// SIMATIC STEP 7 (V5.x) project S_desbobinado
// CPU: CPU312(1)
// station: P_ADR_BUS
// station: Hardware
// station: Equipo SIMATIC 300
// program: Programa S7(1)

SYMBOL_TABLE
"CONTADOR"	C 1	COUNTER
"DESBOBINADO"	FB 1	FB 1	// Función que se encarga del desbobinado
"SENSOR"	I 124.0	BOOL
"PRESENCIA"	I 124.1	BOOL
"BIT_DE_TRABAJO"	I 124.2	BOOL
"START"	I 124.3	BOOL
"STOP"	I 124.4	BOOL
"BAJAR_CONT"	I 124.5	BOOL
"LOAD_CONT"	I 124.6	BOOL
"Cycle Execution"	OB 1	OB 1
"PLANCHAS"	PIW 651	WORD
"CENTRO"	PIW 751	INT
"MCENTRO"	PIW 800	INT
"ABRIRMCENTRO"	Q 100.1	BOOL
"DESBOBINAR"	Q 100.2	BOOL
"BIT_OK"	Q 100.3	BOOL
"BIT_ERROR"	Q 100.4	BOOL
"STBY"	Q 100.5	BOOL
END_SYMBOL_TABLE

FUNCTION_BLOCK "DESBOBINADO"	// FB 1
TITLE = DESBOBINADO
VERSION : 0.1
VAR_INPUT
  SENSOR : BOOL ;
  PRESENCIA : BOOL ;
  CENTRO : INT ;
  bit_de_trabajo : BOOL ;
  MCENTRO : INT ;
  Contador : COUNTER ;
  START : BOOL ;
  PLANCHAS : WORD  := W#16#100;
END_VAR
VAR_OUTPUT
  ABRIRMCENTRO : BOOL ;
  DESBOBINAR : BOOL ;
  STBY : BOOL ;
END_VAR
VAR
  x31 : BOOL ;
  x32 : BOOL ;
  x33 : BOOL ;
  x34 : BOOL ;
  s1 : BOOL ;
  FP_Bit_Tr : BOOL ;
  x30 : BOOL ;
  FP_PRESENCIA : BOOL ;
  FP_BDT : BOOL ;
  FP_START : BOOL ;
END_VAR
VAR_TEMP
  watchdog_master : BOOL ;
END_VAR
BEGIN
NETWORK
TITLE = Arranque
      SET;
      A     #bit_de_trabajo;
      FP    #FP_BDT;
      S     #x30;
      R     #x31;
      R     #x32;
      R     #x33;
      R     #x34;
      R     #s1;
NETWORK
TITLE = x31 a x32
//Comparacion medida centro con medida nominal del centro para pasar de x31 a x32
      A     #x31;
      A(;
      L     #CENTRO;
      L     #MCENTRO;
      ==R;
      );
      R     #x31;
      S     #x32;
NETWORK
TITLE = x32 a x33
//Presencia detecta que la plancha esta en posicion para empezar el proceso de 
//desbobinado-cizallado
      A     #x32;
      A     #PRESENCIA;
      FP    #FP_PRESENCIA;
      R     #x32;
      S     #x33;
NETWORK
TITLE = x33 a x34
//Detecta que la plancha esta lista para ser cizallada
      A     #x33;
      A     #SENSOR;
      R     #x33;
      S     #x34;
NETWORK
TITLE = x34 a x33
//si el contador no ha acabado
      A     #x34;
      T     LD 1;
      TAK;
      T     LD 5;
      L     #Contador;
      T     LW 9;
      L     LD 5;
      L     LD 1;
      A     C [LW 9];
      AN    #SENSOR;
      R     #x34;
      S     #x33;
NETWORK
TITLE = x34 a s1
//si el contador ha cabado
      A     #x34;
      T     LD 1;
      TAK;
      T     LD 5;
      L     #Contador;
      T     LW 9;
      L     LD 5;
      L     LD 1;
      AN    C [LW 9];
      AN    #SENSOR;
      AN    #PRESENCIA;
      R     #x34;
      S     #x30;
NETWORK
TITLE = Tratamiento de bit de fin
      A     #x30;
      =     #STBY;
NETWORK
TITLE = Abrir centro
      A     #x31;
      =     #ABRIRMCENTRO;
NETWORK
TITLE = Carga del contador y desbobinado en x32
      A     #x32;
      S     #DESBOBINAR;
      L     #PLANCHAS;
      T     LD 1;
      TAK;
      T     LD 5;
      L     #Contador;
      T     LW 9;
      L     LD 5;
      L     LD 1;
      S     C [LW 9];
NETWORK
TITLE = Resta del contador y salida del x33
      A     #x33;
      S     #DESBOBINAR;
NETWORK
TITLE =
      A     #x34;
      R     #DESBOBINAR;
NETWORK
TITLE = De X30 a X31
      A     #START;
      FP    #FP_START;
      A     #x30;
      R     #x30;
      S     #x31;
END_FUNCTION_BLOCK

DATA_BLOCK DB 1
VERSION : 0.0
"DESBOBINADO"
BEGIN
END_DATA_BLOCK

ORGANIZATION_BLOCK "Cycle Execution"	// OB 1
TITLE = "Main Program Sweep (Cycle)"
VERSION : 0.1
VAR_TEMP
  OB1_EV_CLASS : BYTE ;	//Bits 0-3 = 1 (Coming event), Bits 4-7 = 1 (Event class 1)
  OB1_SCAN_1 : BYTE ;	//1 (Cold restart scan 1 of OB 1), 3 (Scan 2-n of OB 1)
  OB1_PRIORITY : BYTE ;	//Priority of OB Execution
  OB1_OB_NUMBR : BYTE ;	//1 (Organization block 1, OB1)
  OB1_RESERVED_1 : BYTE ;	//Reserved for system
  OB1_RESERVED_2 : BYTE ;	//Reserved for system
  OB1_PREV_CYCLE : INT ;	//Cycle time of previous OB1 scan (milliseconds)
  OB1_MIN_CYCLE : INT ;	//Minimum cycle time of OB1 (milliseconds)
  OB1_MAX_CYCLE : INT ;	//Maximum cycle time of OB1 (milliseconds)
  OB1_DATE_TIME : DATE_AND_TIME ;	//Date and time OB1 started
END_VAR
BEGIN
NETWORK
TITLE =
      A     "BAJAR_CONT";
      CD    "CONTADOR";
NETWORK
TITLE =
      CALL  "DESBOBINADO" , DB 1 (
           SENSOR                   := "SENSOR",
           PRESENCIA                := "PRESENCIA",
           CENTRO                   := "CENTRO",
           bit_de_trabajo           := "BIT_DE_TRABAJO",
           MCENTRO                  := "MCENTRO",
           Contador                 := "CONTADOR",
           START                    := "START",
           PLANCHAS                 := "PLANCHAS",
           ABRIRMCENTRO             := "ABRIRMCENTRO",
           DESBOBINAR               := "DESBOBINAR",
           STBY                     := "STBY");
END_ORGANIZATION_BLOCK
